PROGRAM MAIN
VAR
END_VAR

SyncProgram();

END_PROGRAM

(* stored: Version 1.1.0.1, ProductVersion 3.1.4024.12
   POU MAIN: Id {c59320b9-08be-403d-80a7-42424e07a971}, SpecialFunc None *)
